(* Logix 5000 project; controller Sucrose_Main Emulate 5570 rev 20.12; software revision 20.01; part 14 of 30 *)
(* tags used below, declared in another part *)
   Alarm_ACK_Master_Timer : TIMER;
   DI_E22_0 : ALIAS FOR FLX_E22:0:I;   // Discrete Input EN2T_FLX 192.168.1.22
   DO_E22_2 : ALIAS FOR FLX_E22:2:O;   // Discrete Output EN2T_FLX 192.168.1.22
   FV230501_AOI : QSI_Flow_Valve;   // FV-23-05-01-O PRE FILTER TRAIN 1 INLET VALVE OPEN
   FV230506_AOI : QSI_Flow_Valve;   // FV-23-05-06-O PRE FILTER TRAIN 1 OUTLET VALVE OPEN
   FV230508_AOI : QSI_Flow_Valve;   // FV-23-05-08-O FINAL FILTER TRAIN 1 INLET VALVE OPEN
   FV230513_AOI : QSI_Flow_Valve;   // FV-23-05-13-O FINAL FILTER TRAIN 1 OUTLET VALVE OPEN
   Rung_Comment : BOOL;
   Sucrose_MM_Enable : BOOL;
   SucroseCIP_FILTRATION_REMOTE : CIP_REMOTE;
   SucroseDischarge : Area_Program;
   SucroseFiltration : Area_Program;
(* FiltrationArea_AutoLogic, continued *)

ROUTINE Enable_Logic_old   (* ladder *)
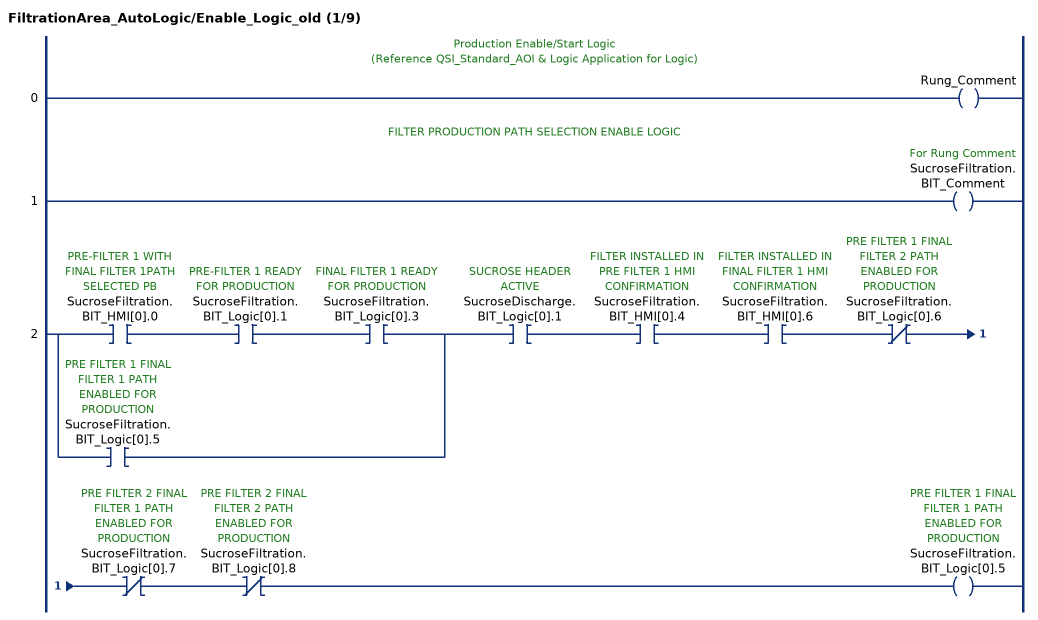
   // Production Enable/Start Logic
   // (Reference QSI_Standard_AOI & Logic Application for Logic)
   0: OTE(Rung_Comment);
   // FILTER PRODUCTION PATH SELECTION ENABLE LOGIC
   1: OTE(SucroseFiltration.BIT_Comment);
   2: [XIC(SucroseFiltration.BIT_HMI[0].0) XIC(SucroseFiltration.BIT_Logic[0].1) XIC(SucroseFiltration.BIT_Logic[0].3) ,XIC(SucroseFiltration.BIT_Logic[0].5) ]XIC(SucroseDischarge.BIT_Logic[0].1)XIC(SucroseFiltration.BIT_HMI[0].4)XIC(SucroseFiltration.BIT_HMI[0].6)XIO(SucroseFiltration.BIT_Logic[0].6)XIO(SucroseFiltration.BIT_Logic[0].7)XIO(SucroseFiltration.BIT_Logic[0].8)OTE(SucroseFiltration.BIT_Logic[0].5);
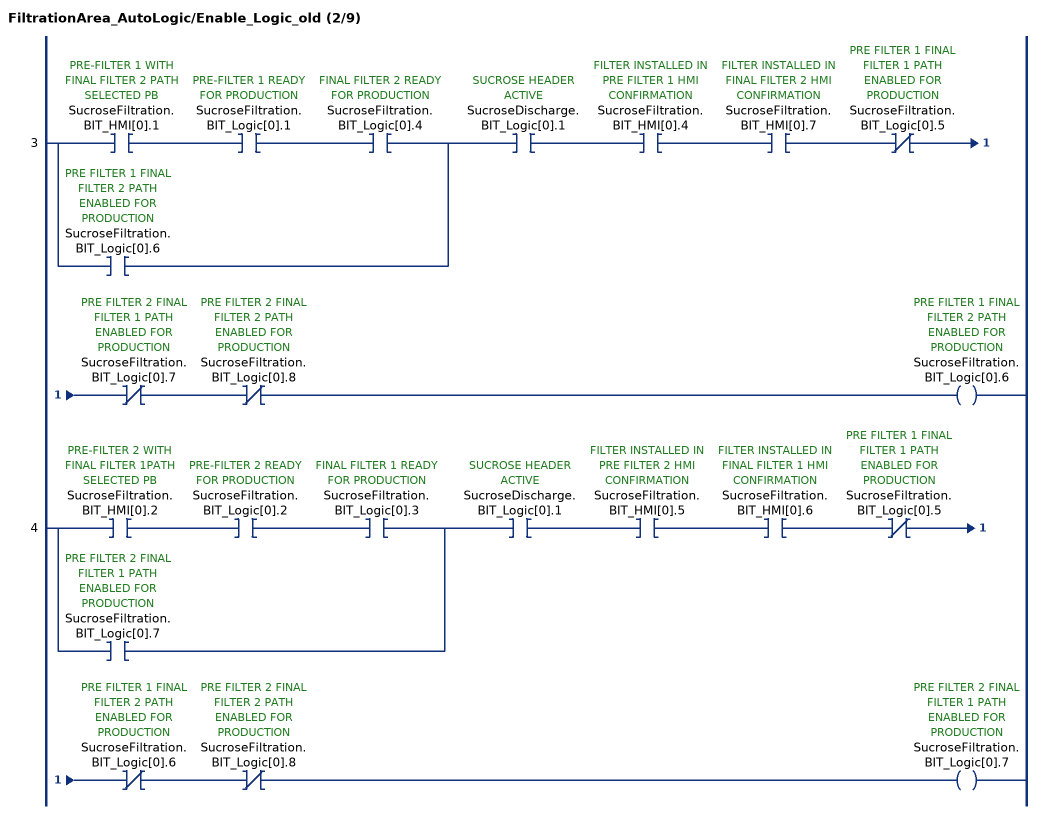
   3: [XIC(SucroseFiltration.BIT_HMI[0].1) XIC(SucroseFiltration.BIT_Logic[0].1) XIC(SucroseFiltration.BIT_Logic[0].4) ,XIC(SucroseFiltration.BIT_Logic[0].6) ]XIC(SucroseDischarge.BIT_Logic[0].1)XIC(SucroseFiltration.BIT_HMI[0].4)XIC(SucroseFiltration.BIT_HMI[0].7)XIO(SucroseFiltration.BIT_Logic[0].5)XIO(SucroseFiltration.BIT_Logic[0].7)XIO(SucroseFiltration.BIT_Logic[0].8)OTE(SucroseFiltration.BIT_Logic[0].6);
   4: [XIC(SucroseFiltration.BIT_HMI[0].2) XIC(SucroseFiltration.BIT_Logic[0].2) XIC(SucroseFiltration.BIT_Logic[0].3) ,XIC(SucroseFiltration.BIT_Logic[0].7) ]XIC(SucroseDischarge.BIT_Logic[0].1)XIC(SucroseFiltration.BIT_HMI[0].5)XIC(SucroseFiltration.BIT_HMI[0].6)XIO(SucroseFiltration.BIT_Logic[0].5)XIO(SucroseFiltration.BIT_Logic[0].6)XIO(SucroseFiltration.BIT_Logic[0].8)OTE(SucroseFiltration.BIT_Logic[0].7);
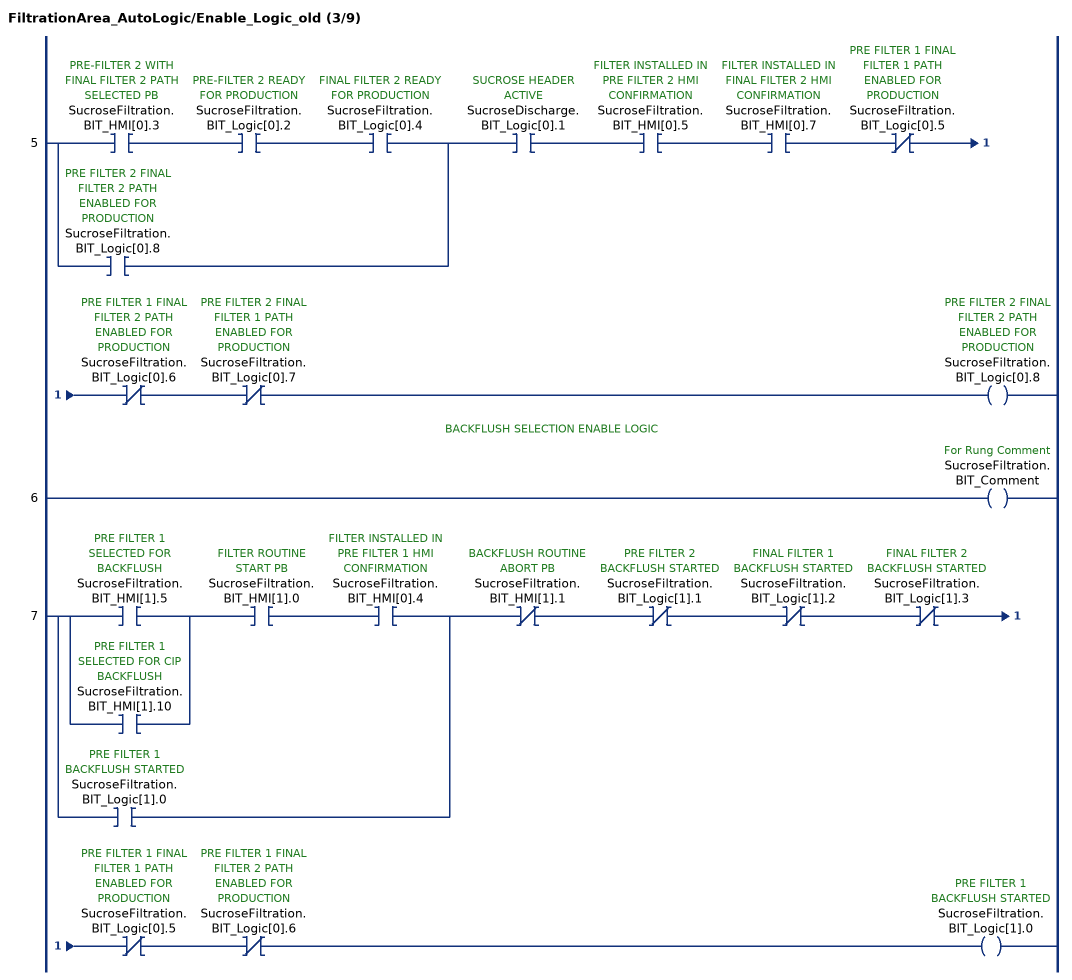
   5: [XIC(SucroseFiltration.BIT_HMI[0].3) XIC(SucroseFiltration.BIT_Logic[0].2) XIC(SucroseFiltration.BIT_Logic[0].4) ,XIC(SucroseFiltration.BIT_Logic[0].8) ]XIC(SucroseDischarge.BIT_Logic[0].1)XIC(SucroseFiltration.BIT_HMI[0].5)XIC(SucroseFiltration.BIT_HMI[0].7)XIO(SucroseFiltration.BIT_Logic[0].5)XIO(SucroseFiltration.BIT_Logic[0].6)XIO(SucroseFiltration.BIT_Logic[0].7)OTE(SucroseFiltration.BIT_Logic[0].8);
   // BACKFLUSH SELECTION ENABLE LOGIC
   6: OTE(SucroseFiltration.BIT_Comment);
   7: [[XIC(SucroseFiltration.BIT_HMI[1].5) ,XIC(SucroseFiltration.BIT_HMI[1].10) ] XIC(SucroseFiltration.BIT_HMI[1].0) XIC(SucroseFiltration.BIT_HMI[0].4) ,XIC(SucroseFiltration.BIT_Logic[1].0) ]XIO(SucroseFiltration.BIT_HMI[1].1)XIO(SucroseFiltration.BIT_Logic[1].1)XIO(SucroseFiltration.BIT_Logic[1].2)XIO(SucroseFiltration.BIT_Logic[1].3)XIO(SucroseFiltration.BIT_Logic[0].5)XIO(SucroseFiltration.BIT_Logic[0].6)OTE(SucroseFiltration.BIT_Logic[1].0);
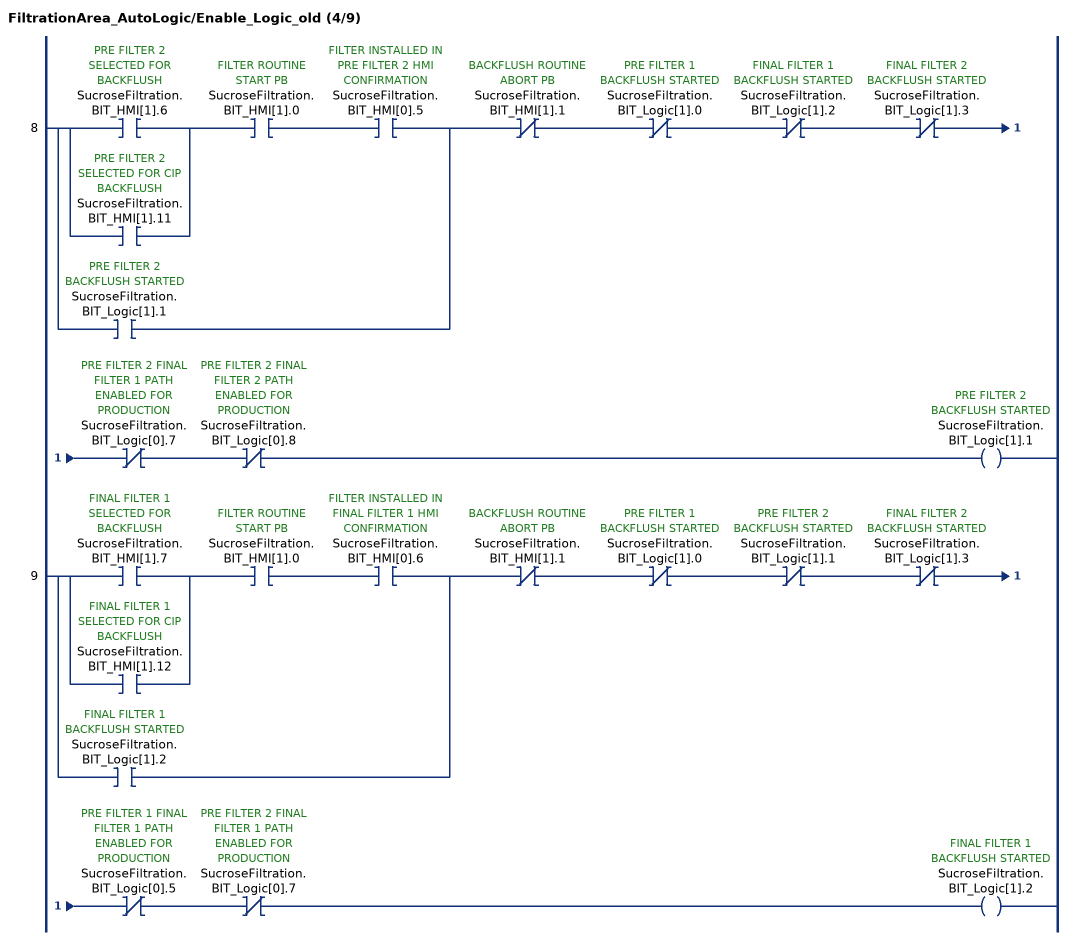
   8: [[XIC(SucroseFiltration.BIT_HMI[1].6) ,XIC(SucroseFiltration.BIT_HMI[1].11) ] XIC(SucroseFiltration.BIT_HMI[1].0) XIC(SucroseFiltration.BIT_HMI[0].5) ,XIC(SucroseFiltration.BIT_Logic[1].1) ]XIO(SucroseFiltration.BIT_HMI[1].1)XIO(SucroseFiltration.BIT_Logic[1].0)XIO(SucroseFiltration.BIT_Logic[1].2)XIO(SucroseFiltration.BIT_Logic[1].3)XIO(SucroseFiltration.BIT_Logic[0].7)XIO(SucroseFiltration.BIT_Logic[0].8)OTE(SucroseFiltration.BIT_Logic[1].1);
   9: [[XIC(SucroseFiltration.BIT_HMI[1].7) ,XIC(SucroseFiltration.BIT_HMI[1].12) ] XIC(SucroseFiltration.BIT_HMI[1].0) XIC(SucroseFiltration.BIT_HMI[0].6) ,XIC(SucroseFiltration.BIT_Logic[1].2) ]XIO(SucroseFiltration.BIT_HMI[1].1)XIO(SucroseFiltration.BIT_Logic[1].0)XIO(SucroseFiltration.BIT_Logic[1].1)XIO(SucroseFiltration.BIT_Logic[1].3)XIO(SucroseFiltration.BIT_Logic[0].5)XIO(SucroseFiltration.BIT_Logic[0].7)OTE(SucroseFiltration.BIT_Logic[1].2);
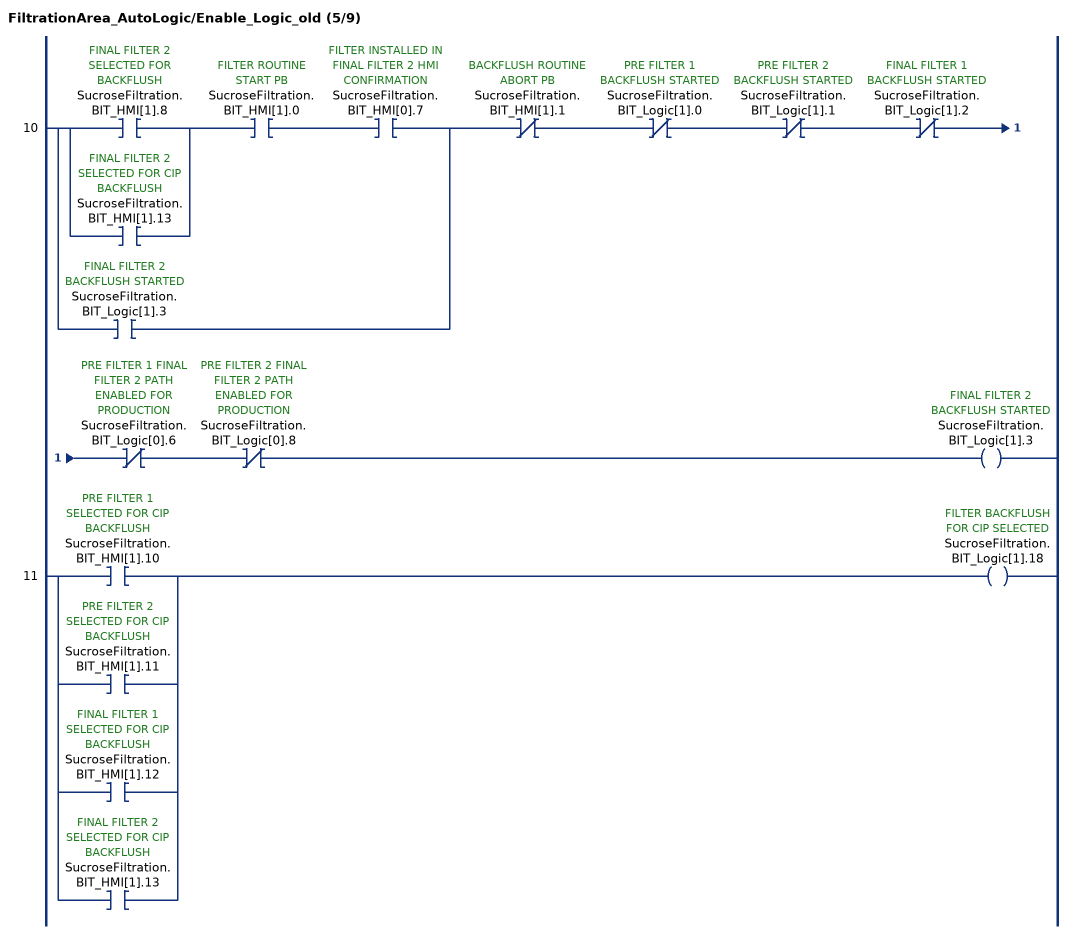
   10: [[XIC(SucroseFiltration.BIT_HMI[1].8) ,XIC(SucroseFiltration.BIT_HMI[1].13) ] XIC(SucroseFiltration.BIT_HMI[1].0) XIC(SucroseFiltration.BIT_HMI[0].7) ,XIC(SucroseFiltration.BIT_Logic[1].3) ]XIO(SucroseFiltration.BIT_HMI[1].1)XIO(SucroseFiltration.BIT_Logic[1].0)XIO(SucroseFiltration.BIT_Logic[1].1)XIO(SucroseFiltration.BIT_Logic[1].2)XIO(SucroseFiltration.BIT_Logic[0].6)XIO(SucroseFiltration.BIT_Logic[0].8)OTE(SucroseFiltration.BIT_Logic[1].3);
   11: [XIC(SucroseFiltration.BIT_HMI[1].10) ,XIC(SucroseFiltration.BIT_HMI[1].11) ,XIC(SucroseFiltration.BIT_HMI[1].12) ,XIC(SucroseFiltration.BIT_HMI[1].13) ]OTE(SucroseFiltration.BIT_Logic[1].18);
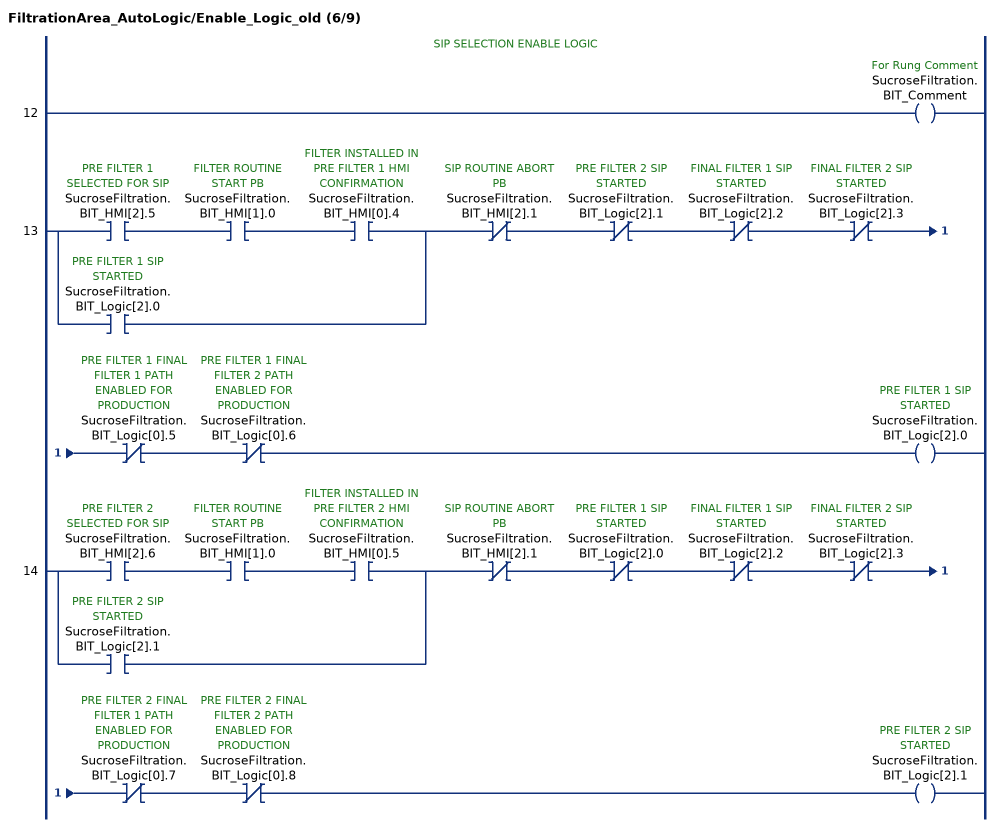
   // SIP SELECTION ENABLE LOGIC
   12: OTE(SucroseFiltration.BIT_Comment);
   13: [XIC(SucroseFiltration.BIT_HMI[2].5) XIC(SucroseFiltration.BIT_HMI[1].0) XIC(SucroseFiltration.BIT_HMI[0].4) ,XIC(SucroseFiltration.BIT_Logic[2].0) ]XIO(SucroseFiltration.BIT_HMI[2].1)XIO(SucroseFiltration.BIT_Logic[2].1)XIO(SucroseFiltration.BIT_Logic[2].2)XIO(SucroseFiltration.BIT_Logic[2].3)XIO(SucroseFiltration.BIT_Logic[0].5)XIO(SucroseFiltration.BIT_Logic[0].6)OTE(SucroseFiltration.BIT_Logic[2].0);
   14: [XIC(SucroseFiltration.BIT_HMI[2].6) XIC(SucroseFiltration.BIT_HMI[1].0) XIC(SucroseFiltration.BIT_HMI[0].5) ,XIC(SucroseFiltration.BIT_Logic[2].1) ]XIO(SucroseFiltration.BIT_HMI[2].1)XIO(SucroseFiltration.BIT_Logic[2].0)XIO(SucroseFiltration.BIT_Logic[2].2)XIO(SucroseFiltration.BIT_Logic[2].3)XIO(SucroseFiltration.BIT_Logic[0].7)XIO(SucroseFiltration.BIT_Logic[0].8)OTE(SucroseFiltration.BIT_Logic[2].1);
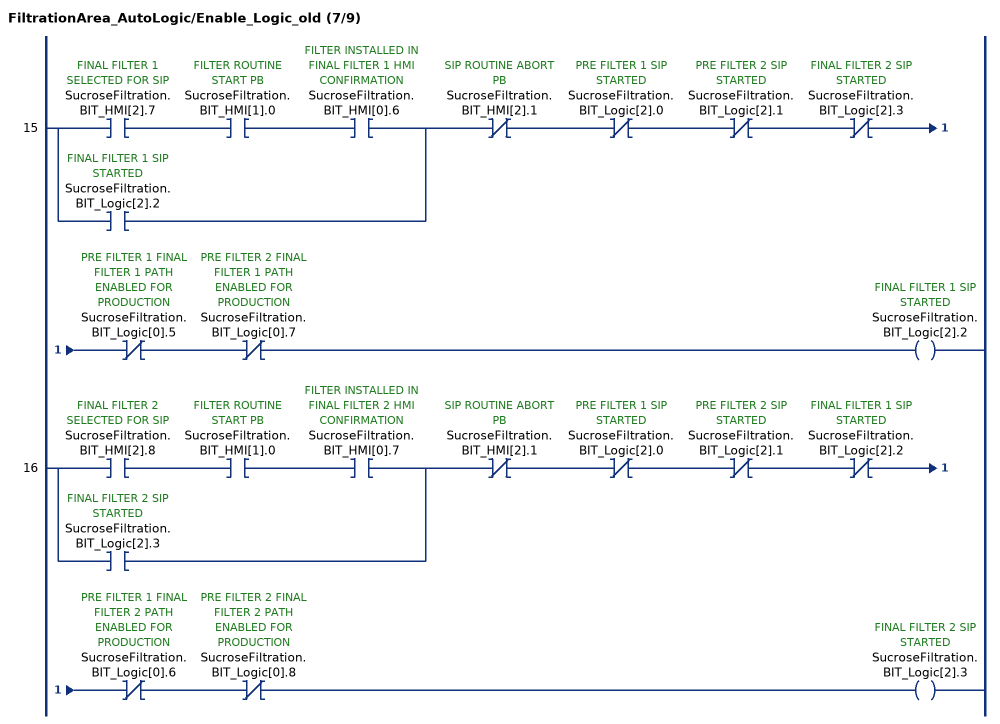
   15: [XIC(SucroseFiltration.BIT_HMI[2].7) XIC(SucroseFiltration.BIT_HMI[1].0) XIC(SucroseFiltration.BIT_HMI[0].6) ,XIC(SucroseFiltration.BIT_Logic[2].2) ]XIO(SucroseFiltration.BIT_HMI[2].1)XIO(SucroseFiltration.BIT_Logic[2].0)XIO(SucroseFiltration.BIT_Logic[2].1)XIO(SucroseFiltration.BIT_Logic[2].3)XIO(SucroseFiltration.BIT_Logic[0].5)XIO(SucroseFiltration.BIT_Logic[0].7)OTE(SucroseFiltration.BIT_Logic[2].2);
   16: [XIC(SucroseFiltration.BIT_HMI[2].8) XIC(SucroseFiltration.BIT_HMI[1].0) XIC(SucroseFiltration.BIT_HMI[0].7) ,XIC(SucroseFiltration.BIT_Logic[2].3) ]XIO(SucroseFiltration.BIT_HMI[2].1)XIO(SucroseFiltration.BIT_Logic[2].0)XIO(SucroseFiltration.BIT_Logic[2].1)XIO(SucroseFiltration.BIT_Logic[2].2)XIO(SucroseFiltration.BIT_Logic[0].6)XIO(SucroseFiltration.BIT_Logic[0].8)OTE(SucroseFiltration.BIT_Logic[2].3);
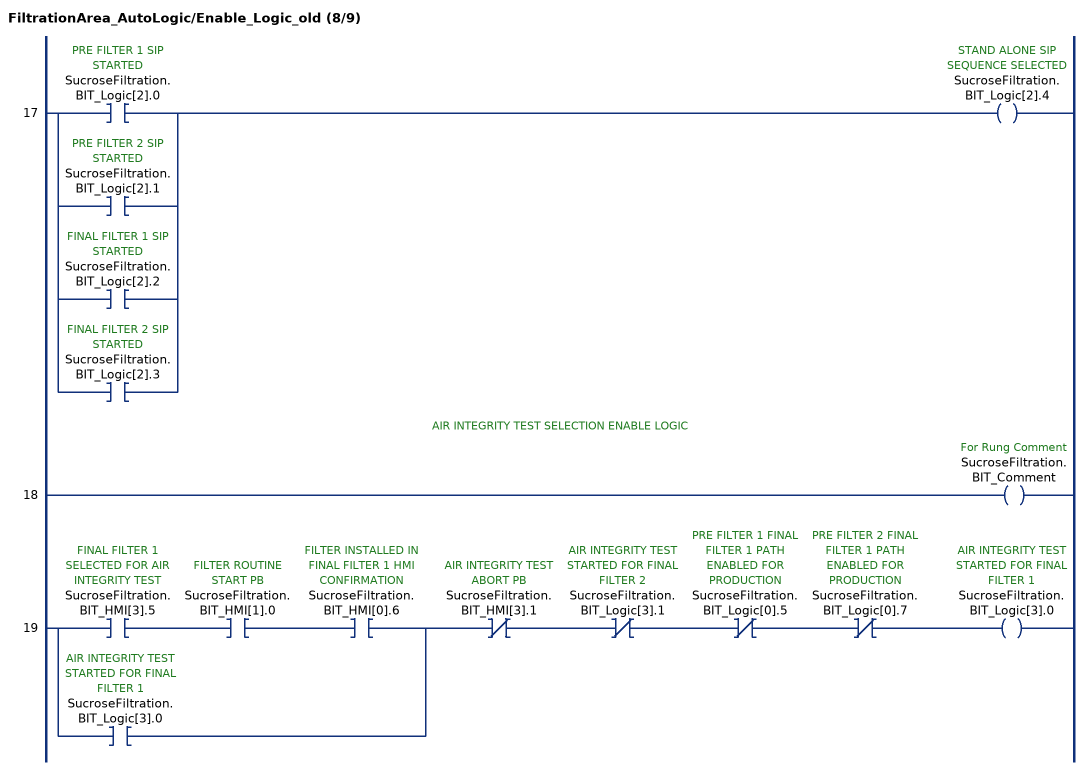
   17: [XIC(SucroseFiltration.BIT_Logic[2].0) ,XIC(SucroseFiltration.BIT_Logic[2].1) ,XIC(SucroseFiltration.BIT_Logic[2].2) ,XIC(SucroseFiltration.BIT_Logic[2].3) ]OTE(SucroseFiltration.BIT_Logic[2].4);
   // AIR INTEGRITY TEST SELECTION ENABLE LOGIC
   18: OTE(SucroseFiltration.BIT_Comment);
   19: [XIC(SucroseFiltration.BIT_HMI[3].5) XIC(SucroseFiltration.BIT_HMI[1].0) XIC(SucroseFiltration.BIT_HMI[0].6) ,XIC(SucroseFiltration.BIT_Logic[3].0) ]XIO(SucroseFiltration.BIT_HMI[3].1)XIO(SucroseFiltration.BIT_Logic[3].1)XIO(SucroseFiltration.BIT_Logic[0].5)XIO(SucroseFiltration.BIT_Logic[0].7)OTE(SucroseFiltration.BIT_Logic[3].0);
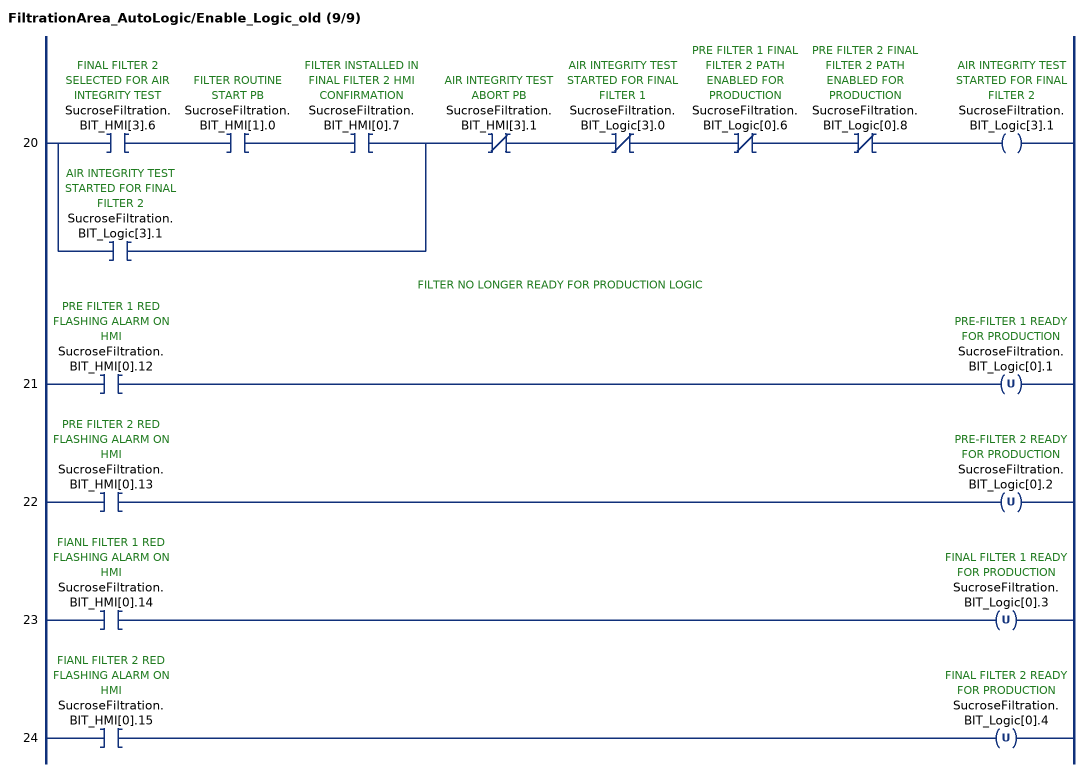
   20: [XIC(SucroseFiltration.BIT_HMI[3].6) XIC(SucroseFiltration.BIT_HMI[1].0) XIC(SucroseFiltration.BIT_HMI[0].7) ,XIC(SucroseFiltration.BIT_Logic[3].1) ]XIO(SucroseFiltration.BIT_HMI[3].1)XIO(SucroseFiltration.BIT_Logic[3].0)XIO(SucroseFiltration.BIT_Logic[0].6)XIO(SucroseFiltration.BIT_Logic[0].8)OTE(SucroseFiltration.BIT_Logic[3].1);
   // FILTER NO LONGER READY FOR PRODUCTION LOGIC
   21: XIC(SucroseFiltration.BIT_HMI[0].12)OTU(SucroseFiltration.BIT_Logic[0].1);
   22: XIC(SucroseFiltration.BIT_HMI[0].13)OTU(SucroseFiltration.BIT_Logic[0].2);
   23: XIC(SucroseFiltration.BIT_HMI[0].14)OTU(SucroseFiltration.BIT_Logic[0].3);
   24: XIC(SucroseFiltration.BIT_HMI[0].15)OTU(SucroseFiltration.BIT_Logic[0].4);
END_ROUTINE

ROUTINE MainRoutine   (* ladder *)
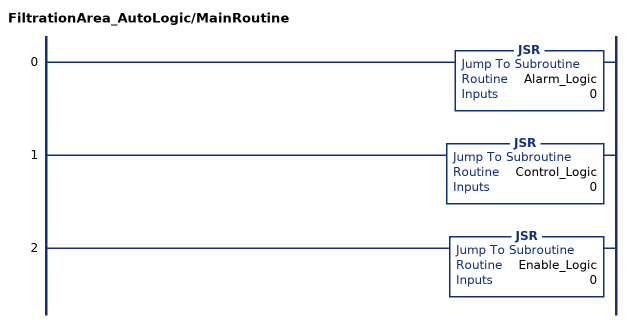
   0: JSR(Alarm_Logic,0);
   1: JSR(Control_Logic,0);
   2: JSR(Enable_Logic,0);
END_ROUTINE
END_PROGRAM

PROGRAM FiltrationArea_EN2T_IO_Discrete_DO_E22_2   (* main routine MainRoutine *)

ROUTINE _00_FV230501   (* ladder *)
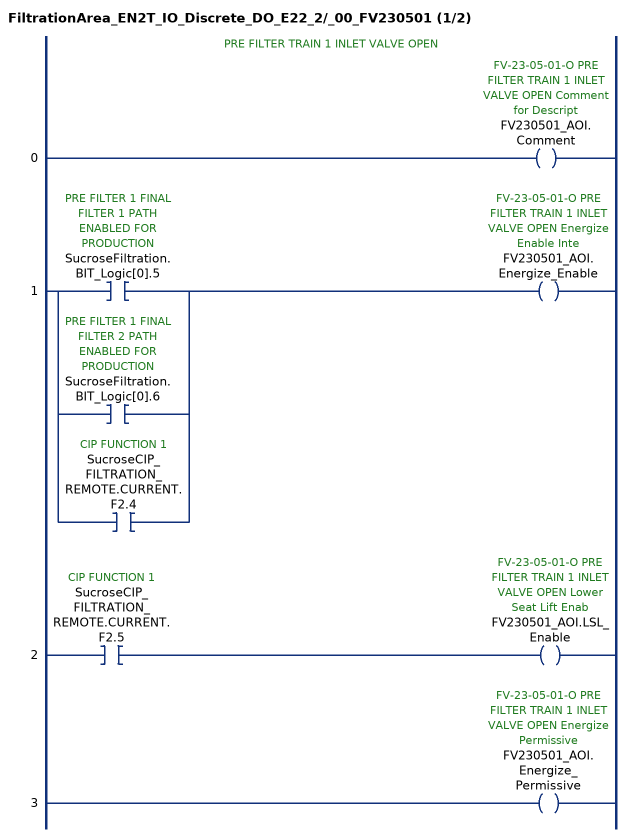
   // PRE FILTER TRAIN 1 INLET VALVE OPEN
   0: OTE(FV230501_AOI.Comment);
   1: [XIC(SucroseFiltration.BIT_Logic[0].5) ,XIC(SucroseFiltration.BIT_Logic[0].6) ,XIC(SucroseCIP_FILTRATION_REMOTE.CURRENT.F2.4) ]OTE(FV230501_AOI.Energize_Enable);
   2: XIC(SucroseCIP_FILTRATION_REMOTE.CURRENT.F2.5)OTE(FV230501_AOI.LSL_Enable);
   3: OTE(FV230501_AOI.Energize_Permissive);
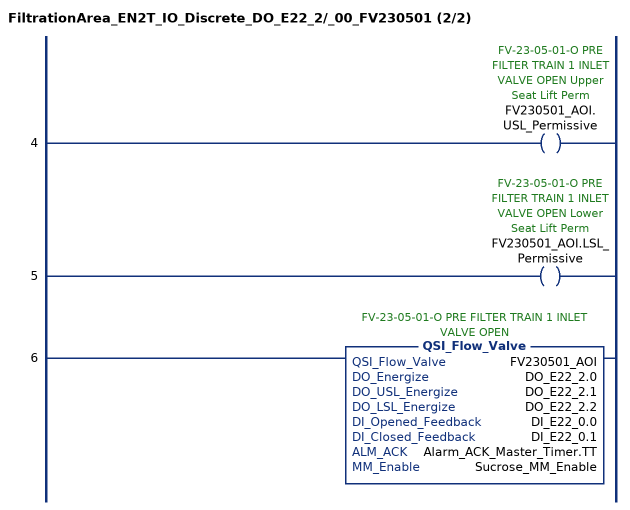
   4: OTE(FV230501_AOI.USL_Permissive);
   5: OTE(FV230501_AOI.LSL_Permissive);
   6: QSI_Flow_Valve(FV230501_AOI,DO_E22_2.0,DO_E22_2.1,DO_E22_2.2,DI_E22_0.0,DI_E22_0.1,Alarm_ACK_Master_Timer.TT,Sucrose_MM_Enable);
END_ROUTINE

ROUTINE _03_FV230506   (* ladder *)
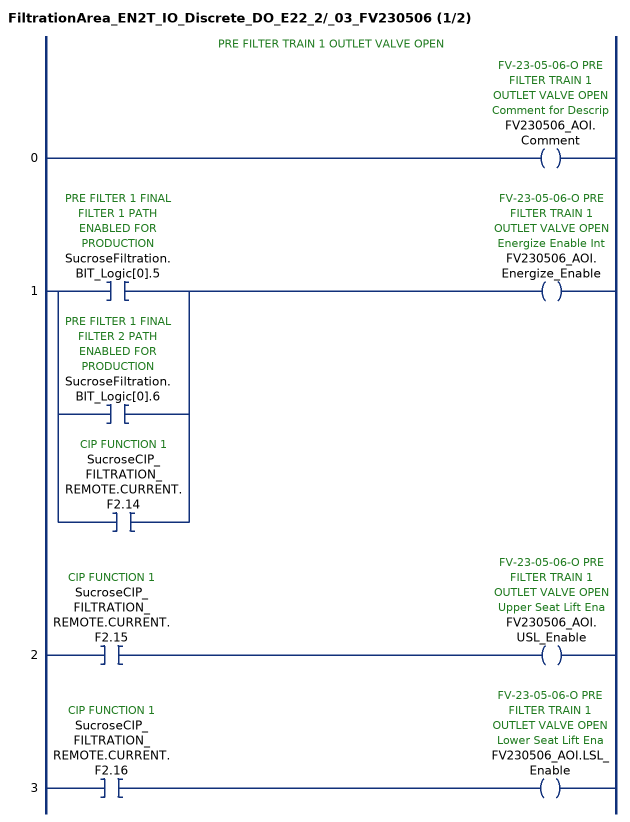
   // PRE FILTER TRAIN 1 OUTLET VALVE OPEN
   0: OTE(FV230506_AOI.Comment);
   1: [XIC(SucroseFiltration.BIT_Logic[0].5) ,XIC(SucroseFiltration.BIT_Logic[0].6) ,XIC(SucroseCIP_FILTRATION_REMOTE.CURRENT.F2.14) ]OTE(FV230506_AOI.Energize_Enable);
   2: XIC(SucroseCIP_FILTRATION_REMOTE.CURRENT.F2.15)OTE(FV230506_AOI.USL_Enable);
   3: XIC(SucroseCIP_FILTRATION_REMOTE.CURRENT.F2.16)OTE(FV230506_AOI.LSL_Enable);
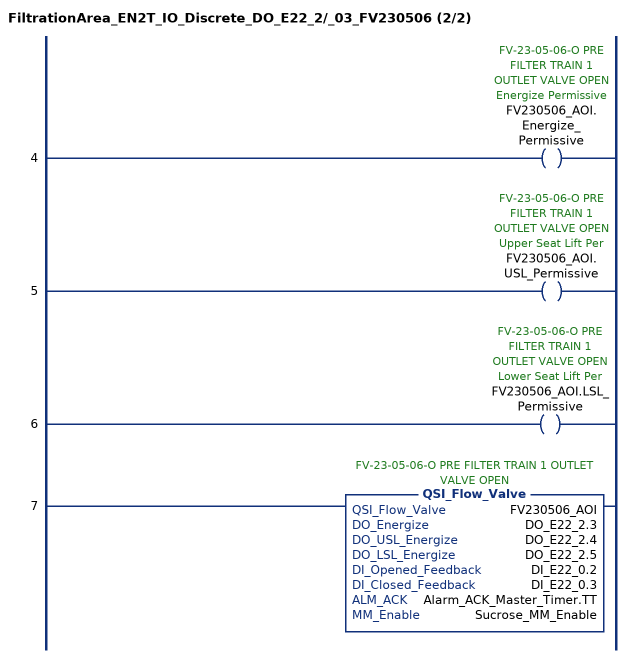
   4: OTE(FV230506_AOI.Energize_Permissive);
   5: OTE(FV230506_AOI.USL_Permissive);
   6: OTE(FV230506_AOI.LSL_Permissive);
   7: QSI_Flow_Valve(FV230506_AOI,DO_E22_2.3,DO_E22_2.4,DO_E22_2.5,DI_E22_0.2,DI_E22_0.3,Alarm_ACK_Master_Timer.TT,Sucrose_MM_Enable);
END_ROUTINE

ROUTINE _06_FV230508   (* ladder *)
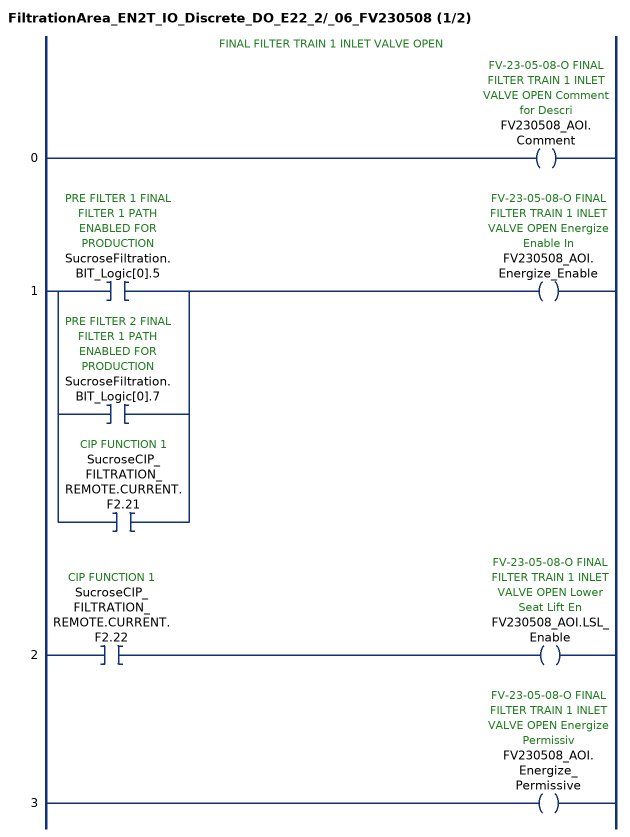
   // FINAL FILTER TRAIN 1 INLET VALVE OPEN
   0: OTE(FV230508_AOI.Comment);
   1: [XIC(SucroseFiltration.BIT_Logic[0].5) ,XIC(SucroseFiltration.BIT_Logic[0].7) ,XIC(SucroseCIP_FILTRATION_REMOTE.CURRENT.F2.21) ]OTE(FV230508_AOI.Energize_Enable);
   2: XIC(SucroseCIP_FILTRATION_REMOTE.CURRENT.F2.22)OTE(FV230508_AOI.LSL_Enable);
   3: OTE(FV230508_AOI.Energize_Permissive);
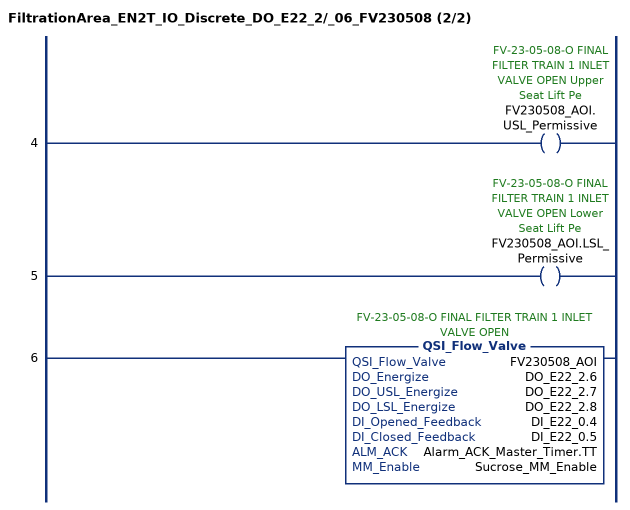
   4: OTE(FV230508_AOI.USL_Permissive);
   5: OTE(FV230508_AOI.LSL_Permissive);
   6: QSI_Flow_Valve(FV230508_AOI,DO_E22_2.6,DO_E22_2.7,DO_E22_2.8,DI_E22_0.4,DI_E22_0.5,Alarm_ACK_Master_Timer.TT,Sucrose_MM_Enable);
END_ROUTINE

ROUTINE _09_FV230513   (* ladder *)
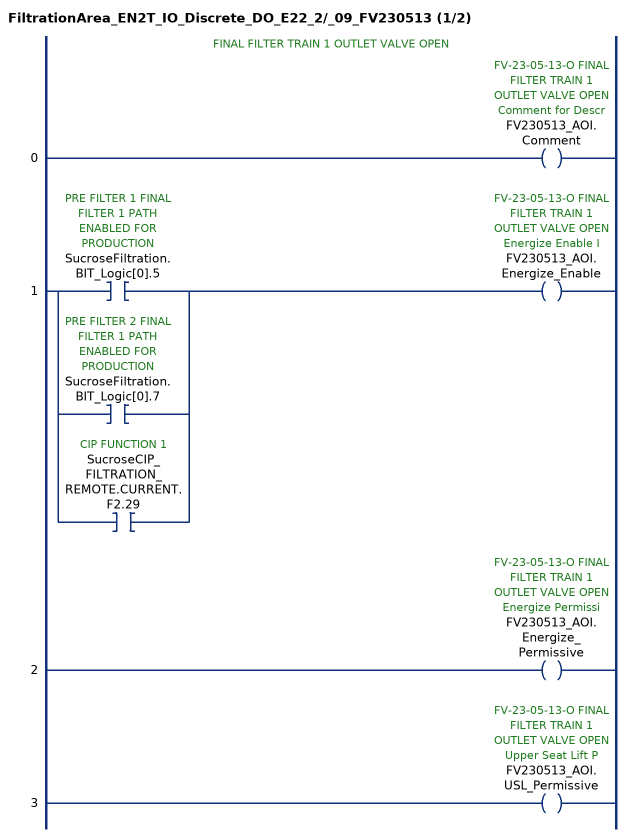
   // FINAL FILTER TRAIN 1 OUTLET VALVE OPEN
   0: OTE(FV230513_AOI.Comment);
   1: [XIC(SucroseFiltration.BIT_Logic[0].5) ,XIC(SucroseFiltration.BIT_Logic[0].7) ,XIC(SucroseCIP_FILTRATION_REMOTE.CURRENT.F2.29) ]OTE(FV230513_AOI.Energize_Enable);
   2: OTE(FV230513_AOI.Energize_Permissive);
   3: OTE(FV230513_AOI.USL_Permissive);
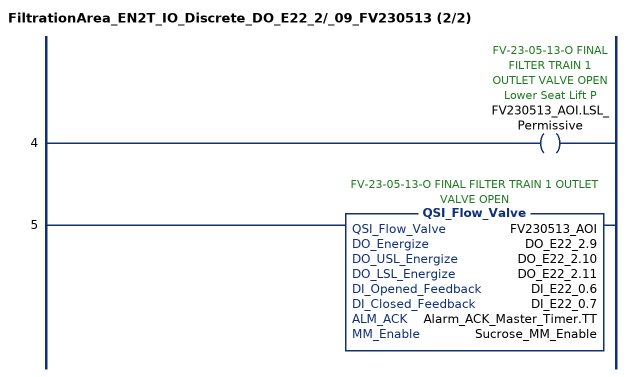
   4: OTE(FV230513_AOI.LSL_Permissive);
   5: QSI_Flow_Valve(FV230513_AOI,DO_E22_2.9,DO_E22_2.10,DO_E22_2.11,DI_E22_0.6,DI_E22_0.7,Alarm_ACK_Master_Timer.TT,Sucrose_MM_Enable);
END_ROUTINE
